FUNCTION F_SafeRelease
VAR_INPUT
	Object : I_Disposable;
END_VAR

IF Object <> 0 THEN
	Object.Release();
END_IF

END_FUNCTION

(* stored: Version 1.1.0.1, ProductVersion 3.1.4024.12
   POU F_SafeRelease: Id {103e1eb7-716e-0044-2f6e-badb145686c4}, SpecialFunc None *)
